// TIA Portal V20 export
DATA_BLOCK "Station_Movikit"   // DB5
{ S7_Optimized_Access := 'TRUE' }
// stored: MemoryReserve 100
   VAR
      MSt34_Fl1_PI : "SEW_MOVIKIT_VelocityDrive_STATUS_V2.1";
      MSt34_Fl1_PO : "SEW_MOVIKIT_VelocityDrive_SETPOINTS_V2.1";
      MSt34_Fl2_PI : "SEW_MOVIKIT_VelocityDrive_STATUS_V2.1";
      MSt34_Fl2_PO : "SEW_MOVIKIT_VelocityDrive_SETPOINTS_V2.1";
      MSt34_Fl3_PI : "SEW_MOVIKIT_VelocityDrive_STATUS_V2.1";
      MSt34_Fl3_PO : "SEW_MOVIKIT_VelocityDrive_SETPOINTS_V2.1";
      MSt34_Fl4_PI : "SEW_MOVIKIT_VelocityDrive_STATUS_V2.1";
      MSt34_Fl4_PO : "SEW_MOVIKIT_VelocityDrive_SETPOINTS_V2.1";
      MSt34_Fl5_PI : "SEW_MOVIKIT_VelocityDrive_STATUS_V2.1";
      MSt34_Fl5_PO : "SEW_MOVIKIT_VelocityDrive_SETPOINTS_V2.1";
      MSt34_Fl6_PI : "SEW_MOVIKIT_VelocityDrive_STATUS_V2.1";
      MSt34_Fl6_PO : "SEW_MOVIKIT_VelocityDrive_SETPOINTS_V2.1";
      MSt32_Fl1_PI : "SEW_MOVIKIT_VelocityDrive_STATUS_V2.1";
      MSt32_Fl1_PO : "SEW_MOVIKIT_VelocityDrive_SETPOINTS_V2.1";
      MSt32_Fl2_PI : "SEW_MOVIKIT_VelocityDrive_STATUS_V2.1";
      MSt32_Fl2_PO : "SEW_MOVIKIT_VelocityDrive_SETPOINTS_V2.1";
      MSt32_Fl3_PI : "SEW_MOVIKIT_VelocityDrive_STATUS_V2.1";
      MSt32_Fl3_PO : "SEW_MOVIKIT_VelocityDrive_SETPOINTS_V2.1";
      MSt32_Fl4_PI : "SEW_MOVIKIT_VelocityDrive_STATUS_V2.1";
      MSt32_Fl4_PO : "SEW_MOVIKIT_VelocityDrive_SETPOINTS_V2.1";
      MSt32_Fl5_PI : "SEW_MOVIKIT_VelocityDrive_STATUS_V2.1";
      MSt32_Fl5_PO : "SEW_MOVIKIT_VelocityDrive_SETPOINTS_V2.1";
      MSt32_Fl6_PI : "SEW_MOVIKIT_VelocityDrive_STATUS_V2.1";
      MSt32_Fl6_PO : "SEW_MOVIKIT_VelocityDrive_SETPOINTS_V2.1";
      MSt31_Fl1_PI : "SEW_MOVIKIT_VelocityDrive_STATUS_V2.1";
      MSt31_Fl1_PO : "SEW_MOVIKIT_VelocityDrive_SETPOINTS_V2.1";
      MSt31_Fl2_PI : "SEW_MOVIKIT_VelocityDrive_STATUS_V2.1";
      MSt31_Fl2_PO : "SEW_MOVIKIT_VelocityDrive_SETPOINTS_V2.1";
      MSt31_Fl3_PI : "SEW_MOVIKIT_VelocityDrive_STATUS_V2.1";
      MSt31_Fl3_PO : "SEW_MOVIKIT_VelocityDrive_SETPOINTS_V2.1";
      MSt31_Fl4_PI : "SEW_MOVIKIT_VelocityDrive_STATUS_V2.1";
      MSt31_Fl4_PO : "SEW_MOVIKIT_VelocityDrive_SETPOINTS_V2.1";
      MSt31_Fl5_PI : "SEW_MOVIKIT_VelocityDrive_STATUS_V2.1";
      MSt31_Fl5_PO : "SEW_MOVIKIT_VelocityDrive_SETPOINTS_V2.1";
      MSt31_Fl6_PI : "SEW_MOVIKIT_VelocityDrive_STATUS_V2.1";
      MSt31_Fl6_PO : "SEW_MOVIKIT_VelocityDrive_SETPOINTS_V2.1";
   END_VAR
BEGIN
END_DATA_BLOCK
